// TIA Portal V18 export
// export: Created 2026-06-08T16:04:38.5744399Z, ExportSetting WithDefaults, DisplayName Totally Integrated Automation Portal, DisplayVersion V18, DisplayName TIA Portal Openness, DisplayVersion V18, DisplayName TIA Portal Version Control Interface, DisplayVersion V18, DisplayName STEP 7 Professional, DisplayVersion V18, DisplayName STEP 7 Safety, DisplayVersion V18, DisplayName WinCC Professional, DisplayVersion V18
FUNCTION "FC_SIMULATION" : Void   // FC4, LAD
{ S7_Optimized_Access := 'TRUE' }
VERSION : 0.1
// stored: AutoNumber true, IsIECCheckEnabled false, SetENOAutomatically false, UDAEnableTagReadback false
   VAR_TEMP   // added for the SCL form of the ladder/FBD networks
      _w1 : Bool;
      _w2 : Bool;
      _w3 : Bool;
      _w4 : Bool;
      _w5 : Bool;
      _w6 : Bool;
   END_VAR
BEGIN

REGION Network 1: KHỞI ĐỘNG LÀ CHẠY SIMU CẢM BIẾN Cao LUÔN
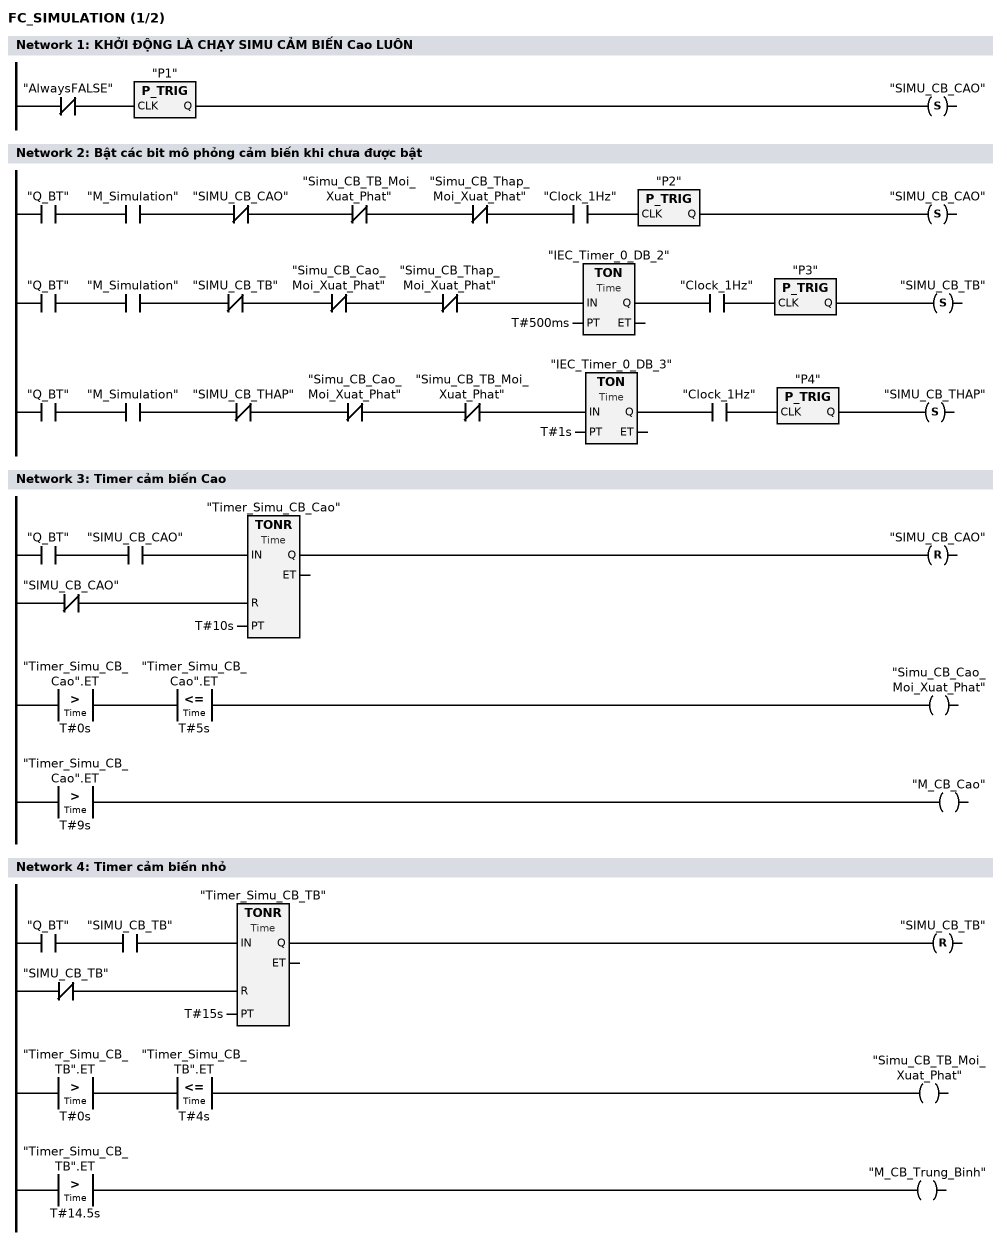
   RUNG wire#powerrail
      I_Contact( "AlwaysFALSE" )
      P_Trig( "P1" )
      S_Coil( "SIMU_CB_CAO" )
   END_RUNG
   // the same network as SCL:
   #_w1 := NOT "AlwaysFALSE" AND NOT "P1";   // rising edge
   "P1" := NOT "AlwaysFALSE";
   IF #_w1 THEN "SIMU_CB_CAO" := TRUE; END_IF;
END_REGION

REGION Network 2: Bật các bit mô phỏng cảm biến khi chưa được bật
   RUNG wire#powerrail
      Contact( "Q_BT" )
      Contact( "M_Simulation" )
      I_Contact( "SIMU_CB_CAO" )
      I_Contact( "Simu_CB_TB_Moi_Xuat_Phat" )
      I_Contact( "Simu_CB_Thap_Moi_Xuat_Phat" )
      Contact( "Clock_1Hz" )
      P_Trig( "P2" )
      S_Coil( "SIMU_CB_CAO" )
   END_RUNG
   RUNG wire#powerrail
      Contact( "Q_BT" )
      Contact( "M_Simulation" )
      I_Contact( "SIMU_CB_TB" )
      I_Contact( "Simu_CB_Cao_Moi_Xuat_Phat" )
      I_Contact( "Simu_CB_Thap_Moi_Xuat_Phat" )
      { S7_Templates := "time_type := Time" } "IEC_Timer_0_DB_2".TON(pt := T#500ms, et =>)
      Contact( "Clock_1Hz" )
      P_Trig( "P3" )
      S_Coil( "SIMU_CB_TB" )
   END_RUNG
   RUNG wire#powerrail
      Contact( "Q_BT" )
      Contact( "M_Simulation" )
      I_Contact( "SIMU_CB_THAP" )
      I_Contact( "Simu_CB_Cao_Moi_Xuat_Phat" )
      I_Contact( "Simu_CB_TB_Moi_Xuat_Phat" )
      { S7_Templates := "time_type := Time" } "IEC_Timer_0_DB_3".TON(pt := T#1s, et =>)
      Contact( "Clock_1Hz" )
      P_Trig( "P4" )
      S_Coil( "SIMU_CB_THAP" )
   END_RUNG
   // the same network as SCL:
   #_w1 := "Q_BT" AND "M_Simulation" AND NOT "SIMU_CB_CAO" AND NOT "Simu_CB_TB_Moi_Xuat_Phat" AND NOT "Simu_CB_Thap_Moi_Xuat_Phat" AND "Clock_1Hz";
   #_w2 := #_w1 AND NOT "P2";   // rising edge
   "P2" := #_w1;
   IF #_w2 THEN "SIMU_CB_CAO" := TRUE; END_IF;
   "IEC_Timer_0_DB_2".TON(IN := "Q_BT" AND "M_Simulation" AND NOT "SIMU_CB_TB" AND NOT "Simu_CB_Cao_Moi_Xuat_Phat" AND NOT "Simu_CB_Thap_Moi_Xuat_Phat",
                          PT := T#500ms);
   #_w3 := "IEC_Timer_0_DB_2".Q AND "Clock_1Hz";
   #_w4 := #_w3 AND NOT "P3";   // rising edge
   "P3" := #_w3;
   IF #_w4 THEN "SIMU_CB_TB" := TRUE; END_IF;
   "IEC_Timer_0_DB_3".TON(IN := "Q_BT" AND "M_Simulation" AND NOT "SIMU_CB_THAP" AND NOT "Simu_CB_Cao_Moi_Xuat_Phat" AND NOT "Simu_CB_TB_Moi_Xuat_Phat",
                          PT := T#1s);
   #_w5 := "IEC_Timer_0_DB_3".Q AND "Clock_1Hz";
   #_w6 := #_w5 AND NOT "P4";   // rising edge
   "P4" := #_w5;
   IF #_w6 THEN "SIMU_CB_THAP" := TRUE; END_IF;
END_REGION

REGION Network 3: Timer cảm biến Cao
   RUNG wire#powerrail
      Contact( "Q_BT" )
      Contact( "SIMU_CB_CAO" )
      { S7_Templates := "time_type := Time" } "Timer_Simu_CB_Cao".TONR(r := wire#w1, pt := T#10s, et =>)
      R_Coil( "SIMU_CB_CAO" )
   END_RUNG
   RUNG wire#powerrail
      I_Contact( "SIMU_CB_CAO" )
   END_RUNG wire#w1
   RUNG wire#powerrail
      { S7_Templates := "SrcType := Time" } GT_Contact(in1 := "Timer_Simu_CB_Cao".ET, in2 := T#0s)
      { S7_Templates := "SrcType := Time" } LE_Contact(in1 := "Timer_Simu_CB_Cao".ET, in2 := T#5s)
      Coil( "Simu_CB_Cao_Moi_Xuat_Phat" )
   END_RUNG
   RUNG wire#powerrail
      { S7_Templates := "SrcType := Time" } GT_Contact(in1 := "Timer_Simu_CB_Cao".ET, in2 := T#9s)
      Coil( "M_CB_Cao" )
   END_RUNG
   // the same network as SCL:
   "Timer_Simu_CB_Cao".TONR(IN := "Q_BT" AND "SIMU_CB_CAO", R := NOT "SIMU_CB_CAO", PT := T#10s);
   IF "Timer_Simu_CB_Cao".Q THEN "SIMU_CB_CAO" := FALSE; END_IF;
   "Simu_CB_Cao_Moi_Xuat_Phat" := ("Timer_Simu_CB_Cao".ET > T#0s) AND ("Timer_Simu_CB_Cao".ET <= T#5s);
   "M_CB_Cao" := "Timer_Simu_CB_Cao".ET > T#9s;
END_REGION

REGION Network 4: Timer cảm biến nhỏ
   RUNG wire#powerrail
      Contact( "Q_BT" )
      Contact( "SIMU_CB_TB" )
      { S7_Templates := "time_type := Time" } "Timer_Simu_CB_TB".TONR(r := wire#w1, pt := T#15s, et =>)
      R_Coil( "SIMU_CB_TB" )
   END_RUNG
   RUNG wire#powerrail
      I_Contact( "SIMU_CB_TB" )
   END_RUNG wire#w1
   RUNG wire#powerrail
      { S7_Templates := "SrcType := Time" } GT_Contact(in1 := "Timer_Simu_CB_TB".ET, in2 := T#0s)
      { S7_Templates := "SrcType := Time" } LE_Contact(in1 := "Timer_Simu_CB_TB".ET, in2 := T#4s)
      Coil( "Simu_CB_TB_Moi_Xuat_Phat" )
   END_RUNG
   RUNG wire#powerrail
      { S7_Templates := "SrcType := Time" } GT_Contact(in1 := "Timer_Simu_CB_TB".ET, in2 := T#14.5s)
      Coil( "M_CB_Trung_Binh" )
   END_RUNG
   // the same network as SCL:
   "Timer_Simu_CB_TB".TONR(IN := "Q_BT" AND "SIMU_CB_TB", R := NOT "SIMU_CB_TB", PT := T#15s);
   IF "Timer_Simu_CB_TB".Q THEN "SIMU_CB_TB" := FALSE; END_IF;
   "Simu_CB_TB_Moi_Xuat_Phat" := ("Timer_Simu_CB_TB".ET > T#0s) AND ("Timer_Simu_CB_TB".ET <= T#4s);
   "M_CB_Trung_Binh" := "Timer_Simu_CB_TB".ET > T#14.5s;
END_REGION

REGION Network 5: Mô phỏng cảm biến trung bình
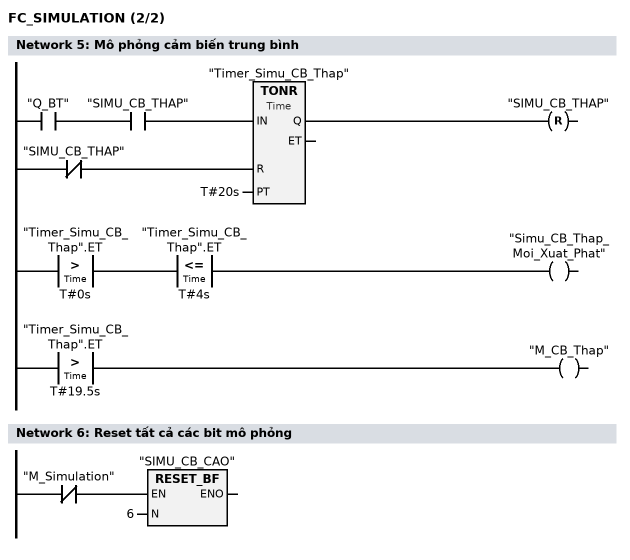
   RUNG wire#powerrail
      Contact( "Q_BT" )
      Contact( "SIMU_CB_THAP" )
      { S7_Templates := "time_type := Time" } "Timer_Simu_CB_Thap".TONR(r := wire#w1, pt := T#20s, et =>)
      R_Coil( "SIMU_CB_THAP" )
   END_RUNG
   RUNG wire#powerrail
      I_Contact( "SIMU_CB_THAP" )
   END_RUNG wire#w1
   RUNG wire#powerrail
      { S7_Templates := "SrcType := Time" } GT_Contact(in1 := "Timer_Simu_CB_Thap".ET, in2 := T#0s)
      { S7_Templates := "SrcType := Time" } LE_Contact(in1 := "Timer_Simu_CB_Thap".ET, in2 := T#4s)
      Coil( "Simu_CB_Thap_Moi_Xuat_Phat" )
   END_RUNG
   RUNG wire#powerrail
      { S7_Templates := "SrcType := Time" } GT_Contact(in1 := "Timer_Simu_CB_Thap".ET, in2 := T#19.5s)
      Coil( "M_CB_Thap" )
   END_RUNG
   // the same network as SCL:
   "Timer_Simu_CB_Thap".TONR(IN := "Q_BT" AND "SIMU_CB_THAP", R := NOT "SIMU_CB_THAP", PT := T#20s);
   IF "Timer_Simu_CB_Thap".Q THEN "SIMU_CB_THAP" := FALSE; END_IF;
   "Simu_CB_Thap_Moi_Xuat_Phat" := ("Timer_Simu_CB_Thap".ET > T#0s) AND ("Timer_Simu_CB_Thap".ET <= T#4s);
   "M_CB_Thap" := "Timer_Simu_CB_Thap".ET > T#19.5s;
END_REGION

REGION Network 6: Reset tất cả các bit mô phỏng
   // no SCL statement known for RBitfield: written as a call
   IF NOT "M_Simulation" THEN RESET_BF(operand := "SIMU_CB_CAO", n := 6); END_IF;
END_REGION
END_FUNCTION
